Fanuc KAREL source: SET_ATTR_PRG.kl

PROGRAM T
%NOLOCKGROUP
VAR
 v0 : STRING[40]
 v1 : INTEGER
 v2 : INTEGER
 v3 : STRING[40]
 v4 : INTEGER
BEGIN
 SET_ATTR_PRG(v0, v1, v2, v3, v4)
END T
